{attribute 'qualified_only'}
TYPE E_MMPathState :
(
	eMMPathState_Initialization 		:= 0,																		(**)
	eMMPathState_Startup				:= 1,																		(**)
	eMMPathState_Operational			:= 2,																		(**)
	eMMPathState_ResetInProgress		:= 3,																		(**)
	eMMPathState_ProgrammingInProgress	:= 4																		(**)
) BYTE;
END_TYPE

(* stored: Version 1.1.0.1, ProductVersion 3.1.4024.5
   EnumerationTextList E_MMPathState: Id {bf6e63a2-0301-4f17-8ce6-78c906f70abd} *)
